// TIA Portal V20 export
TYPE "typeSequenceControlNodeJobInterface_GRnR"
// stored: Namespace Unit1.Em5
   STRUCT
      transferPnPLeft : "Unit1.Em5.typeSequenceControlNodetransferPnPLeftJobInterface_GRnR";
      transferPnPRight : "Unit1.Em5.typeSequenceControlNodetransferPnPRightJobInterface_GRnR";
   END_STRUCT;
END_TYPE
